// TIA Portal V18 export
// export: Created 2026-06-24T03:56:38.1819955Z, ExportSetting WithDefaults, DisplayName Totally Integrated Automation Portal, DisplayVersion V18, DisplayName TIA Portal Openness, DisplayVersion V18, DisplayName TIA Portal Version Control Interface, DisplayVersion V18, DisplayName STEP 7 Professional, DisplayVersion V18, DisplayName STEP 7 Safety, DisplayVersion V18, DisplayName WinCC Professional, DisplayVersion V18
FUNCTION_BLOCK "PID"   // FB1, SCL
{ S7_Optimized_Access := 'TRUE' }
VERSION : 0.1
// stored: AutoNumber true, IsIECCheckEnabled false, IsRetainMemResEnabled false, MemoryReserve 100, SetENOAutomatically false, UDAEnableTagReadback false
   VAR_INPUT
      ki : Real := 0.002;
      kp : Real := 11.0;
      kd : Real;
      level : Real;
      setpoint : Real;
      drain : Bool;
      "full drain" : Bool;
      emergency : Bool;
   END_VAR
   VAR_OUTPUT
      filling : Real;
      draining : Real;
      errordisplay : Real;
      setpointdisplay : DInt;
      leveldisplay : DInt;
   END_VAR
   VAR
      integralop : Real;
      oldintegral : Real;
      err2 : Real;
   END_VAR
   VAR_TEMP
      error : Real;
      u : Real;
      temp : DInt;
   END_VAR
BEGIN

   #errordisplay := ABS(#setpoint - #level);

   //display setpoint to 100%
   #setpointdisplay := REAL_TO_DINT(#setpoint*10.0);
   //



   //display level to 100%
   #leveldisplay :=REAL_TO_DINT( #level*10.0);
   //
   #temp := REAL_TO_DINT(#kp);

   #error := #setpoint - #level;

   #integralop := #integralop + #error; //sums all the past errors to present error
   #u := (#error * #kp) + (#integralop * (#ki / 10)) + (#kd * (#err2 - #error));
   #filling := #u;
   #draining := -#u;


   //if error always goes up the filling will always goes up
   //and it will be more that 100% .but the valve can go only to 100% open
   //so if it goes up.we stop the valve at 10 and  stabilized the integral
   IF (#filling > 10.0) THEN
       #integralop := #oldintegral;
       #filling := 10.0;
   END_IF;
   //same thing but for values under 0
   IF (#filling < 0.0) THEN
       #integralop := #oldintegral;
       #filling := 0.0;
   END_IF;
   IF (#draining > 10.0) THEN
       #integralop := #oldintegral;
       #draining := 10.0;
   END_IF;

   IF (#draining < 0.0) THEN
       #integralop := #oldintegral;
       #draining := 0.0;
   END_IF;

   #oldintegral := #integralop; //past error sum
   #err2 := #error;//past error

   IF #drain THEN
       #draining := 10.0;

   END_IF;

   IF #"full drain" THEN
       #draining := 10.0;
       #filling := 0;
   END_IF;
   IF #emergency THEN
       #draining := 0;
       #filling := 0;

   END_IF;
END_FUNCTION_BLOCK
